{attribute 'GeneratedUsingTerminal: AT2050-0500-0024'}
{attribute addProperty BoxType "AT2050-0500-0024"}
{attribute addProperty Id "A_0089_AT2050_5501_0018_AT2050_5501AT2050_33A3DF1B80"}
{attribute addProperty CRC "2369953933"}
{attribute addProperty Size "80"}
{attribute addProperty Name "A_0055(AT2050-0500-0024)"}
TYPE A_0055_AT2050_0500_0024_8D42A08D EXTENDS AT2050_2EA6C9BF :
STRUCT
	{attribute addProperty Name "A_0089(AT2050-5501-0018) (AT2050-5501)"}
	{attribute addProperty PreviousPort "A_0055(AT2050-0500-0024) : B"}
	A_0089_AT2050_5501_0018_AT2050_5501 : AT2050_33A3DF1B;
END_STRUCT
END_TYPE

(* stored: Version 1.2.0.0, ProductVersion 3.1.4024.11
   DUT A_0055_AT2050_0500_0024_8D42A08D: Id {c80edbe2-fa37-4764-ac08-183fdd1b868a} *)
